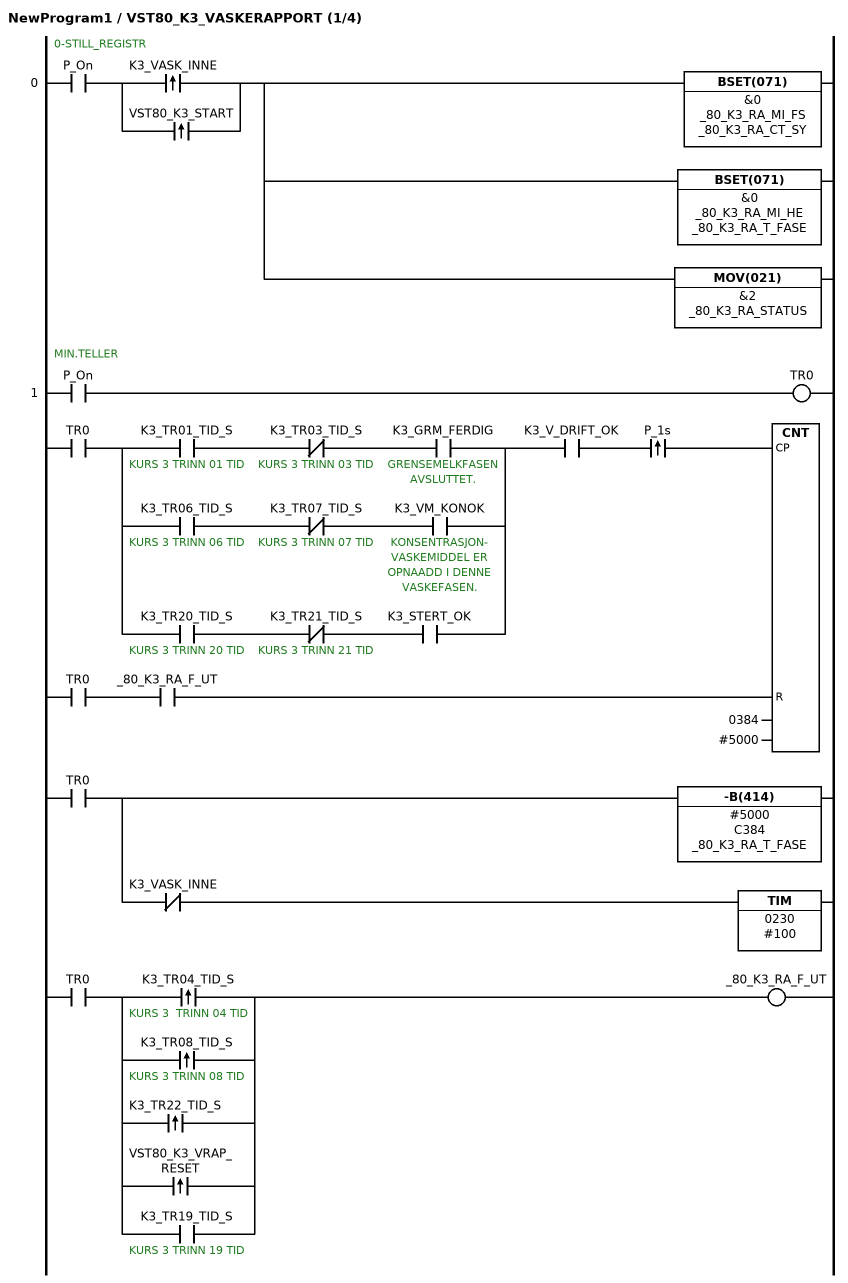
; [picture p384: NewProgram1 / VST80_K3_VASKERAPPORT, rungs 0-1]
; rung 0: 0-STILL_REGISTR
LD P_On
@LD K3_VASK_INNE
@OR VST80_K3_START
ANDLD
BSET(071) &0 _80_K3_RA_MI_FS _80_K3_RA_CT_SY
BSET(071) &0 _80_K3_RA_MI_HE _80_K3_RA_T_FASE
MOV(021) &2 _80_K3_RA_STATUS
; rung 1: MIN.TELLER
LD P_On
OUT TR0
LD K3_TR01_TID_S  ; KURS 3 TRINN 01 TID
ANDNOT K3_TR03_TID_S  ; KURS 3 TRINN 03 TID
AND K3_GRM_FERDIG  ; GRENSEMELKFASEN AVSLUTTET.
LD K3_TR06_TID_S  ; KURS 3 TRINN 06 TID
ANDNOT K3_TR07_TID_S  ; KURS 3 TRINN 07 TID
AND K3_VM_KONOK  ; KONSENTRASJON-VASKEMIDDEL ER OPNAADD I DENNE VASKEFASEN.
ORLD
LD K3_TR20_TID_S  ; KURS 3 TRINN 20 TID
ANDNOT K3_TR21_TID_S  ; KURS 3 TRINN 21 TID
AND K3_STERT_OK
ORLD
ANDLD
AND K3_V_DRIFT_OK
@AND P_1s
LD TR0
AND _80_K3_RA_F_UT
CNT 0384 #5000
LD TR0
-B(414) #5000 C384 _80_K3_RA_T_FASE
ANDNOT K3_VASK_INNE
TIM 0230 #100
LD TR0
@LD K3_TR04_TID_S  ; KURS 3  TRINN 04 TID
@OR K3_TR08_TID_S  ; KURS 3 TRINN 08 TID
@OR K3_TR22_TID_S
@OR VST80_K3_VRAP_RESET
OR K3_TR19_TID_S  ; KURS 3 TRINN 19 TID
ANDLD
OUT _80_K3_RA_F_UT

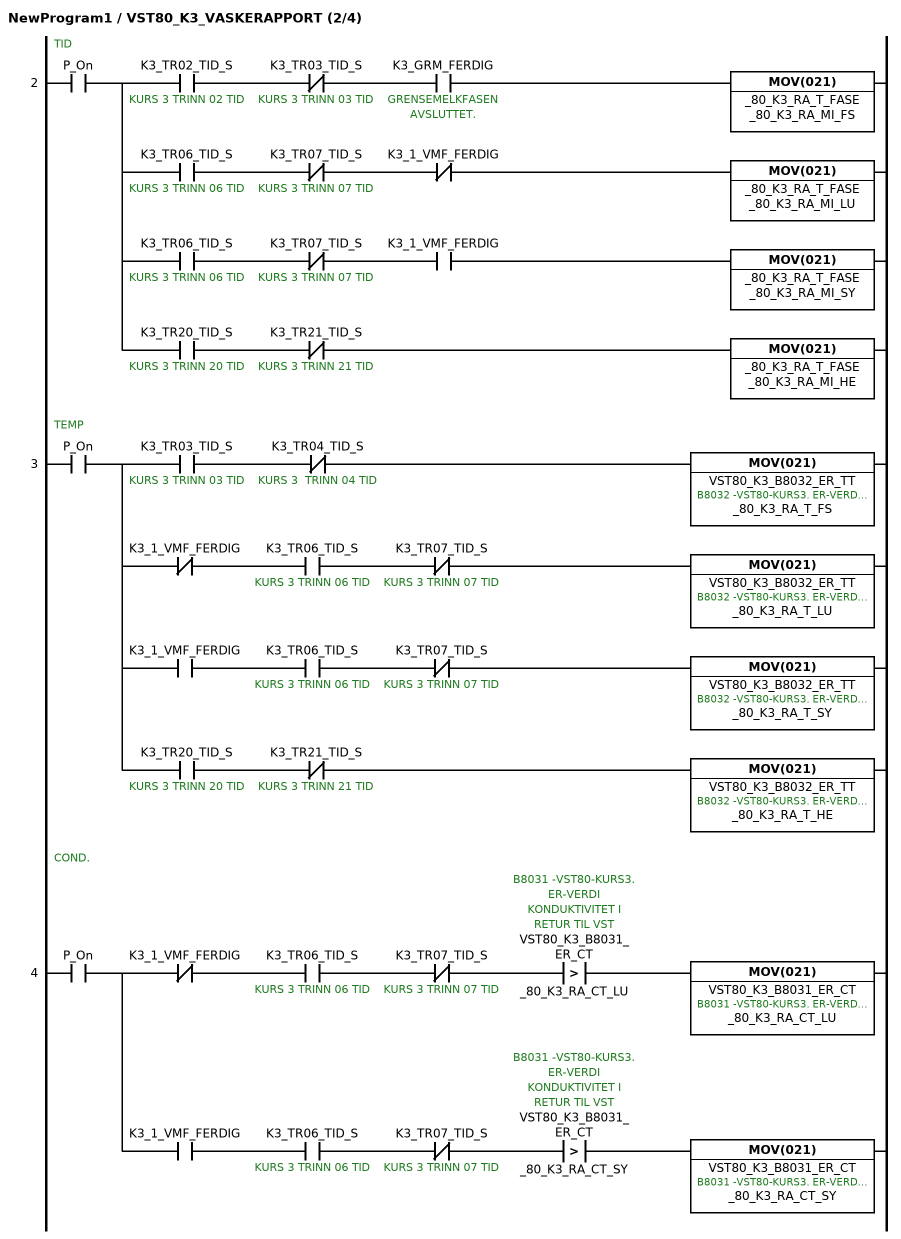
; rung 2: TID
LD P_On
OUT TR0
AND K3_TR02_TID_S  ; KURS 3 TRINN 02 TID
ANDNOT K3_TR03_TID_S  ; KURS 3 TRINN 03 TID
AND K3_GRM_FERDIG  ; GRENSEMELKFASEN AVSLUTTET.
MOV(021) _80_K3_RA_T_FASE _80_K3_RA_MI_FS
LD TR0
AND K3_TR06_TID_S  ; KURS 3 TRINN 06 TID
ANDNOT K3_TR07_TID_S  ; KURS 3 TRINN 07 TID
ANDNOT K3_1_VMF_FERDIG
MOV(021) _80_K3_RA_T_FASE _80_K3_RA_MI_LU
LD TR0
AND K3_TR06_TID_S  ; KURS 3 TRINN 06 TID
ANDNOT K3_TR07_TID_S  ; KURS 3 TRINN 07 TID
AND K3_1_VMF_FERDIG
MOV(021) _80_K3_RA_T_FASE _80_K3_RA_MI_SY
LD TR0
AND K3_TR20_TID_S  ; KURS 3 TRINN 20 TID
ANDNOT K3_TR21_TID_S  ; KURS 3 TRINN 21 TID
MOV(021) _80_K3_RA_T_FASE _80_K3_RA_MI_HE
; rung 3: TEMP
LD P_On
OUT TR0
AND K3_TR03_TID_S  ; KURS 3 TRINN 03 TID
ANDNOT K3_TR04_TID_S  ; KURS 3  TRINN 04 TID
MOV(021) VST80_K3_B8032_ER_TT _80_K3_RA_T_FS  ; B8032 -VST80-KURS3. ER-VERDI TEMPERATUR I RETUR TIL VST
LD TR0
ANDNOT K3_1_VMF_FERDIG
AND K3_TR06_TID_S  ; KURS 3 TRINN 06 TID
ANDNOT K3_TR07_TID_S  ; KURS 3 TRINN 07 TID
MOV(021) VST80_K3_B8032_ER_TT _80_K3_RA_T_LU  ; B8032 -VST80-KURS3. ER-VERDI TEMPERATUR I RETUR TIL VST
LD TR0
AND K3_1_VMF_FERDIG
AND K3_TR06_TID_S  ; KURS 3 TRINN 06 TID
ANDNOT K3_TR07_TID_S  ; KURS 3 TRINN 07 TID
MOV(021) VST80_K3_B8032_ER_TT _80_K3_RA_T_SY  ; B8032 -VST80-KURS3. ER-VERDI TEMPERATUR I RETUR TIL VST
LD TR0
AND K3_TR20_TID_S  ; KURS 3 TRINN 20 TID
ANDNOT K3_TR21_TID_S  ; KURS 3 TRINN 21 TID
MOV(021) VST80_K3_B8032_ER_TT _80_K3_RA_T_HE  ; B8032 -VST80-KURS3. ER-VERDI TEMPERATUR I RETUR TIL VST
; rung 4: COND.
LD P_On
OUT TR0
ANDNOT K3_1_VMF_FERDIG
AND K3_TR06_TID_S  ; KURS 3 TRINN 06 TID
ANDNOT K3_TR07_TID_S  ; KURS 3 TRINN 07 TID
AND>(320) VST80_K3_B8031_ER_CT _80_K3_RA_CT_LU  ; B8031 -VST80-KURS3. ER-VERDI KONDUKTIVITET I RETUR TIL VST
MOV(021) VST80_K3_B8031_ER_CT _80_K3_RA_CT_LU  ; B8031 -VST80-KURS3. ER-VERDI KONDUKTIVITET I RETUR TIL VST
LD TR0
AND K3_1_VMF_FERDIG
AND K3_TR06_TID_S  ; KURS 3 TRINN 06 TID
ANDNOT K3_TR07_TID_S  ; KURS 3 TRINN 07 TID
AND>(320) VST80_K3_B8031_ER_CT _80_K3_RA_CT_SY  ; B8031 -VST80-KURS3. ER-VERDI KONDUKTIVITET I RETUR TIL VST
MOV(021) VST80_K3_B8031_ER_CT _80_K3_RA_CT_SY  ; B8031 -VST80-KURS3. ER-VERDI KONDUKTIVITET I RETUR TIL VST

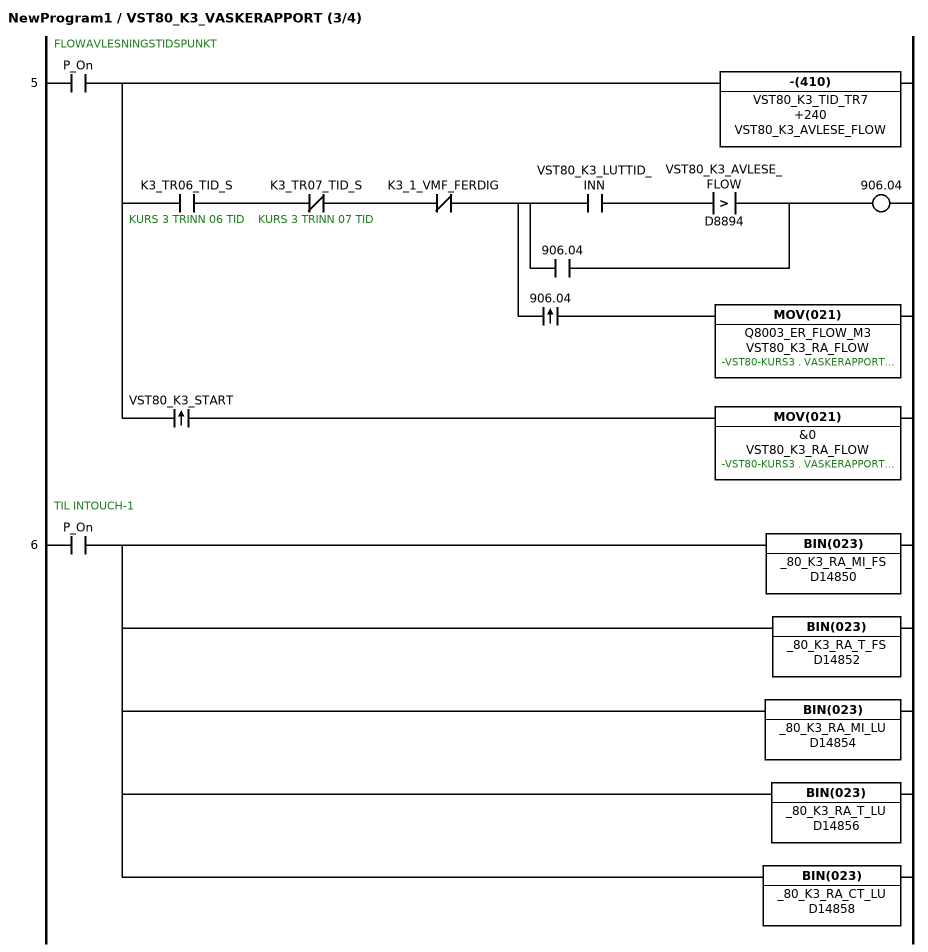
; rung 5: FLOWAVLESNINGSTIDSPUNKT
LD P_On
OUT TR0
-(410) VST80_K3_TID_TR7 +240 VST80_K3_AVLESE_FLOW
AND K3_TR06_TID_S  ; KURS 3 TRINN 06 TID
ANDNOT K3_TR07_TID_S  ; KURS 3 TRINN 07 TID
ANDNOT K3_1_VMF_FERDIG
OUT TR1
LD VST80_K3_LUTTID_INN
AND>(320) VST80_K3_AVLESE_FLOW D8894
OR 906.04
ANDLD
OUT 906.04
LD TR1
@AND 906.04
MOV(021) Q8003_ER_FLOW_M3 VST80_K3_RA_FLOW  ; -VST80-KURS3 . VASKERAPPORT.  FLOW
LD TR0
@AND VST80_K3_START
MOV(021) &0 VST80_K3_RA_FLOW  ; -VST80-KURS3 . VASKERAPPORT.  FLOW
; rung 6: TIL INTOUCH-1
LD P_On
BIN(023) _80_K3_RA_MI_FS D14850
BIN(023) _80_K3_RA_T_FS D14852
BIN(023) _80_K3_RA_MI_LU D14854
BIN(023) _80_K3_RA_T_LU D14856
BIN(023) _80_K3_RA_CT_LU D14858

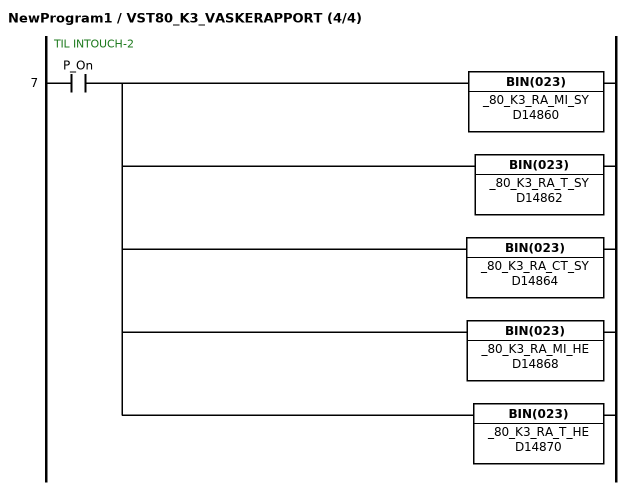
; rung 7: TIL INTOUCH-2
LD P_On
BIN(023) _80_K3_RA_MI_SY D14860
BIN(023) _80_K3_RA_T_SY D14862
BIN(023) _80_K3_RA_CT_SY D14864
BIN(023) _80_K3_RA_MI_HE D14868
BIN(023) _80_K3_RA_T_HE D14870
; rung 8: Ingen_kommentar_funnet

### Section VST80_K3_REGULATORER

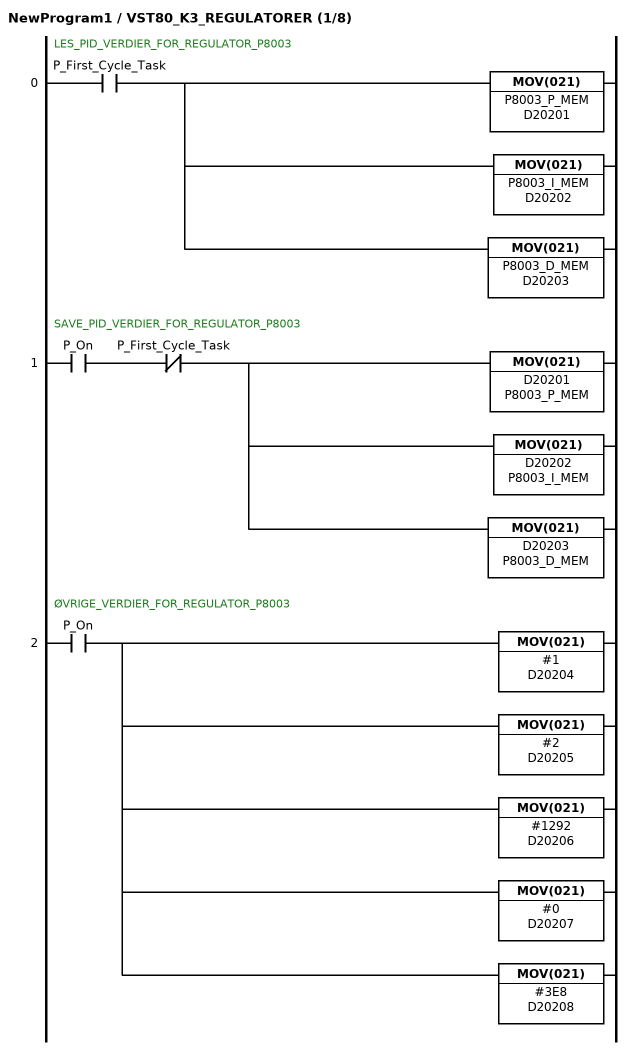
; rung 0: LES_PID_VERDIER_FOR_REGULATOR_P8003
LD P_First_Cycle_Task
MOV(021) P8003_P_MEM D20201
MOV(021) P8003_I_MEM D20202
MOV(021) P8003_D_MEM D20203
; rung 1: SAVE_PID_VERDIER_FOR_REGULATOR_P8003
LD P_On
ANDNOT P_First_Cycle_Task
MOV(021) D20201 P8003_P_MEM
MOV(021) D20202 P8003_I_MEM
MOV(021) D20203 P8003_D_MEM
; rung 2: ØVRIGE_VERDIER_FOR_REGULATOR_P8003
LD P_On
MOV(021) #1 D20204
MOV(021) #2 D20205
MOV(021) #1292 D20206
MOV(021) #0 D20207
MOV(021) #3E8 D20208

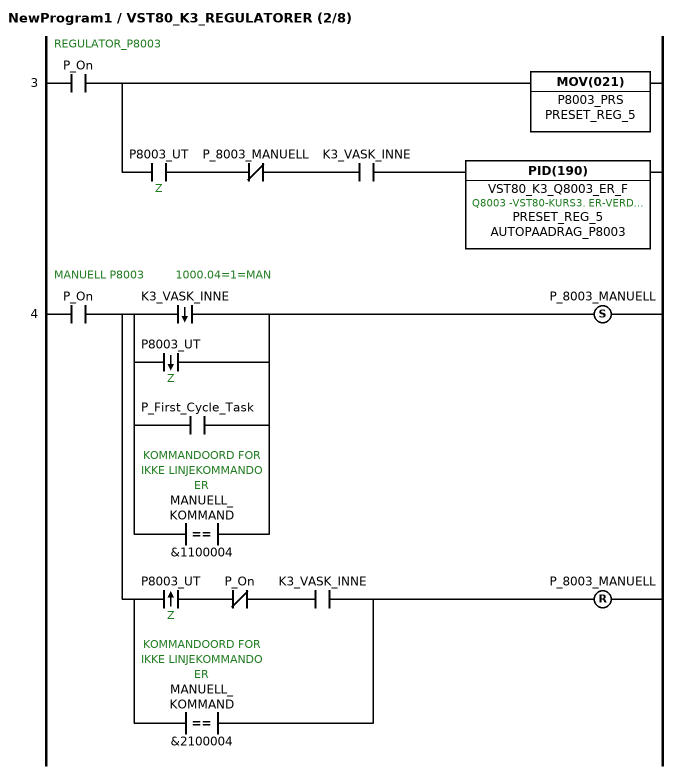
; rung 3: REGULATOR_P8003
LD P_On
MOV(021) P8003_PRS PRESET_REG_5
AND P8003_UT  ; Z
ANDNOT P_8003_MANUELL
AND K3_VASK_INNE
PID(190) VST80_K3_Q8003_ER_F PRESET_REG_5 AUTOPAADRAG_P8003  ; Q8003 -VST80-KURS3. ER-VERDI FLOW I TUR
; rung 4: MANUELL P8003         1000.04=1=MAN
LD P_On
OUT TR0
%LD K3_VASK_INNE
%OR P8003_UT  ; Z
OR P_First_Cycle_Task
OR=L(301) MANUELL_KOMMAND &1100004  ; KOMMANDOORD FOR IKKE LINJEKOMMANDOER
ANDLD
SET P_8003_MANUELL
LD TR0
@LD P8003_UT  ; Z
ANDNOT P_On
AND K3_VASK_INNE
OR=L(301) MANUELL_KOMMAND &2100004  ; KOMMANDOORD FOR IKKE LINJEKOMMANDOER
ANDLD
RSET P_8003_MANUELL

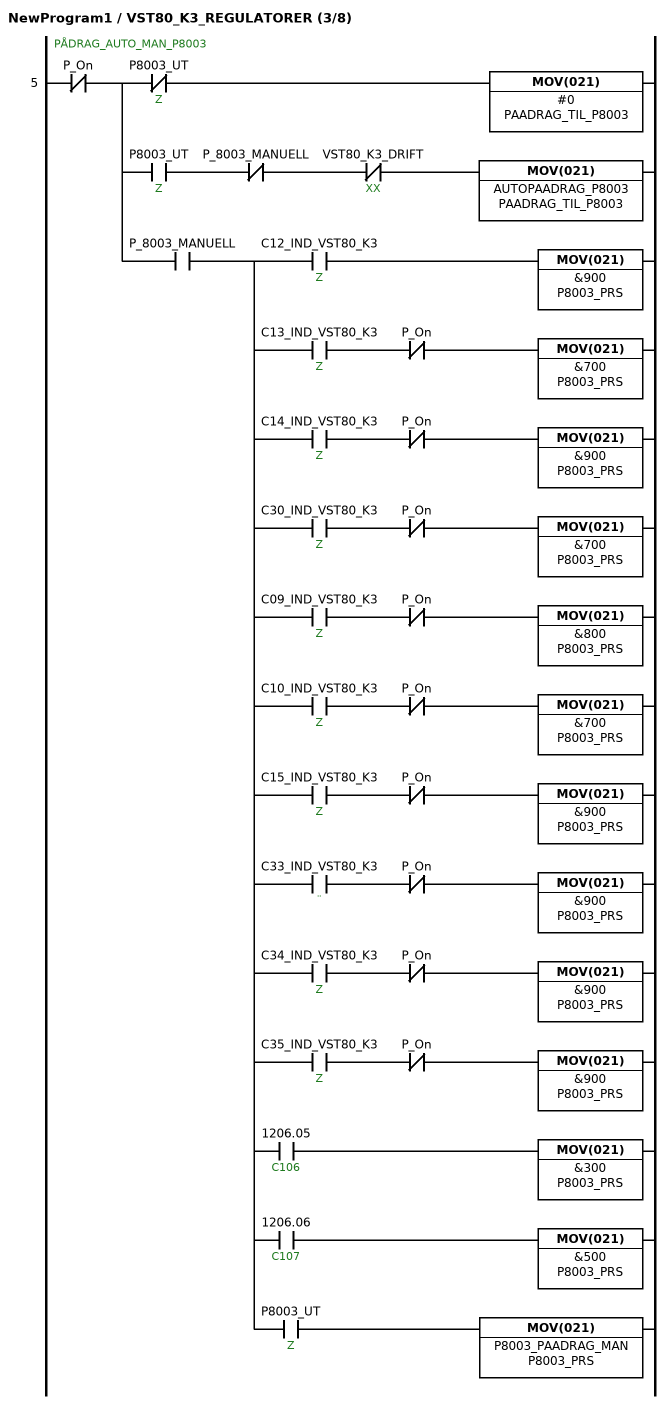
; rung 5: PÅDRAG_AUTO_MAN_P8003
LDNOT P_On
OUT TR0
ANDNOT P8003_UT  ; Z
MOV(021) #0 PAADRAG_TIL_P8003
LD TR0
AND P8003_UT  ; Z
ANDNOT P_8003_MANUELL
ANDNOT VST80_K3_DRIFT  ; XX
MOV(021) AUTOPAADRAG_P8003 PAADRAG_TIL_P8003
LD TR0
AND P_8003_MANUELL
OUT TR0
AND C12_IND_VST80_K3  ; Z
MOV(021) &900 P8003_PRS
LD TR0
AND C13_IND_VST80_K3  ; Z
ANDNOT P_On
MOV(021) &700 P8003_PRS
LD TR0
AND C14_IND_VST80_K3  ; Z
ANDNOT P_On
MOV(021) &900 P8003_PRS
LD TR0
AND C30_IND_VST80_K3  ; Z
ANDNOT P_On
MOV(021) &700 P8003_PRS
LD TR0
AND C09_IND_VST80_K3  ; Z
ANDNOT P_On
MOV(021) &800 P8003_PRS
LD TR0
AND C10_IND_VST80_K3  ; Z
ANDNOT P_On
MOV(021) &700 P8003_PRS
LD TR0
AND C15_IND_VST80_K3  ; Z
ANDNOT P_On
MOV(021) &900 P8003_PRS
LD TR0
AND C33_IND_VST80_K3  ; ¨
ANDNOT P_On
MOV(021) &900 P8003_PRS
LD TR0
AND C34_IND_VST80_K3  ; Z
ANDNOT P_On
MOV(021) &900 P8003_PRS
LD TR0
AND C35_IND_VST80_K3  ; Z
ANDNOT P_On
MOV(021) &900 P8003_PRS
LD TR0
AND 1206.05  ; C106
MOV(021) &300 P8003_PRS
LD TR0
AND 1206.06  ; C107
MOV(021) &500 P8003_PRS
LD TR0
AND P8003_UT  ; Z
MOV(021) P8003_PAADRAG_MAN P8003_PRS

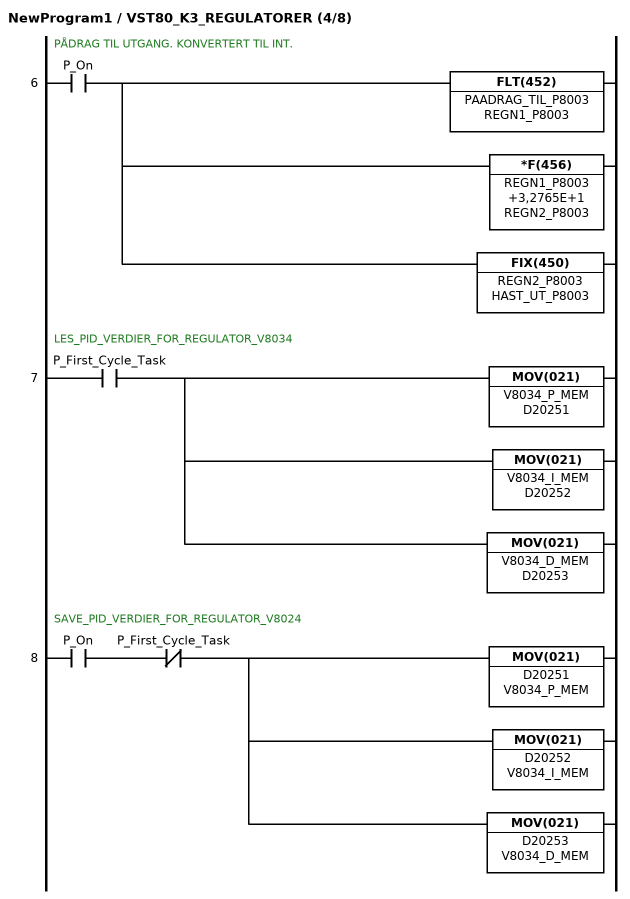
; rung 6: PÅDRAG TIL UTGANG. KONVERTERT TIL INT.
LD P_On
FLT(452) PAADRAG_TIL_P8003 REGN1_P8003
*F(456) REGN1_P8003 +3,2765E+1 REGN2_P8003
FIX(450) REGN2_P8003 HAST_UT_P8003
; rung 7: LES_PID_VERDIER_FOR_REGULATOR_V8034
LD P_First_Cycle_Task
MOV(021) V8034_P_MEM D20251
MOV(021) V8034_I_MEM D20252
MOV(021) V8034_D_MEM D20253
; rung 8: SAVE_PID_VERDIER_FOR_REGULATOR_V8024
LD P_On
ANDNOT P_First_Cycle_Task
MOV(021) D20251 V8034_P_MEM
MOV(021) D20252 V8034_I_MEM
MOV(021) D20253 V8034_D_MEM

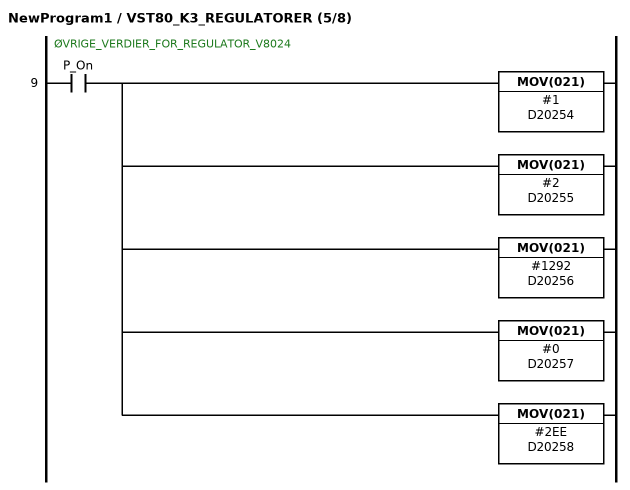
; rung 9: ØVRIGE_VERDIER_FOR_REGULATOR_V8024
LD P_On
MOV(021) #1 D20254
MOV(021) #2 D20255
MOV(021) #1292 D20256
MOV(021) #0 D20257
MOV(021) #2EE D20258

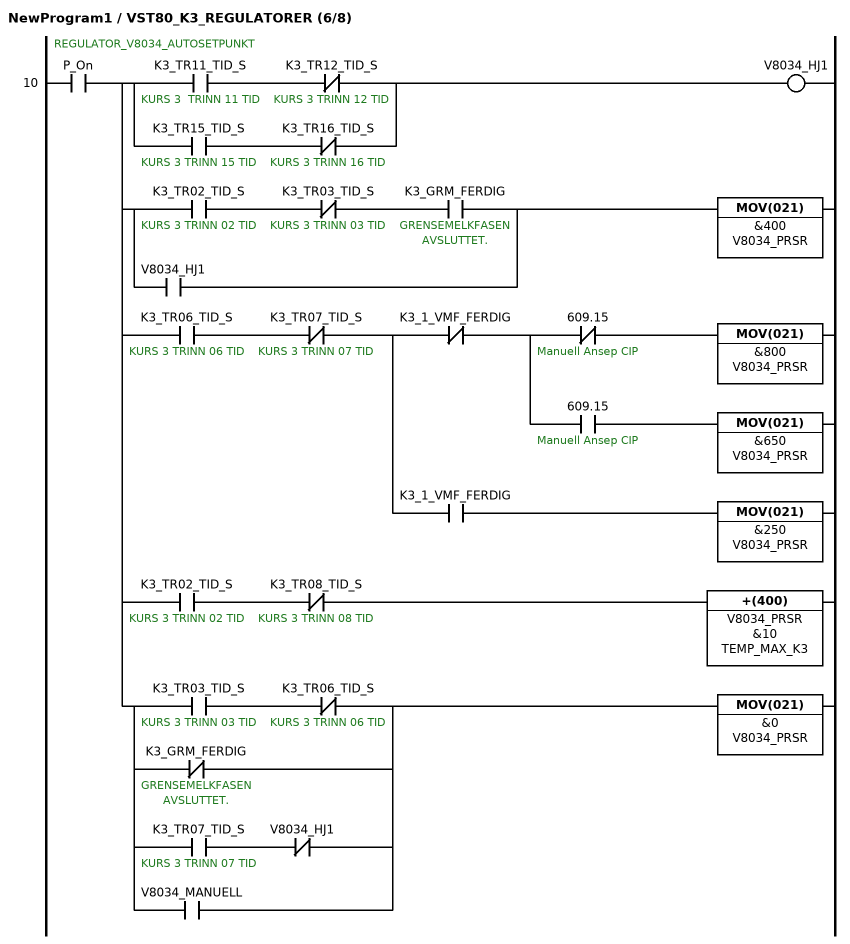
; rung 10: REGULATOR_V8034_AUTOSETPUNKT
LD P_On
OUT TR0
LD K3_TR11_TID_S  ; KURS 3  TRINN 11 TID
ANDNOT K3_TR12_TID_S  ; KURS 3 TRINN 12 TID
LD K3_TR15_TID_S  ; KURS 3 TRINN 15 TID
ANDNOT K3_TR16_TID_S  ; KURS 3 TRINN 16 TID
ORLD
ANDLD
OUT V8034_HJ1
LD TR0
LD K3_TR02_TID_S  ; KURS 3 TRINN 02 TID
ANDNOT K3_TR03_TID_S  ; KURS 3 TRINN 03 TID
AND K3_GRM_FERDIG  ; GRENSEMELKFASEN AVSLUTTET.
OR V8034_HJ1
ANDLD
MOV(021) &400 V8034_PRSR
LD TR0
AND K3_TR06_TID_S  ; KURS 3 TRINN 06 TID
ANDNOT K3_TR07_TID_S  ; KURS 3 TRINN 07 TID
OUT TR1
ANDNOT K3_1_VMF_FERDIG
OUT TR2
ANDNOT 609.15  ; Manuell Ansep CIP
MOV(021) &800 V8034_PRSR
LD TR2
AND 609.15  ; Manuell Ansep CIP
MOV(021) &650 V8034_PRSR
LD TR1
AND K3_1_VMF_FERDIG
MOV(021) &250 V8034_PRSR
LD TR0
AND K3_TR02_TID_S  ; KURS 3 TRINN 02 TID
ANDNOT K3_TR08_TID_S  ; KURS 3 TRINN 08 TID
+(400) V8034_PRSR &10 TEMP_MAX_K3
LD TR0
LD K3_TR03_TID_S  ; KURS 3 TRINN 03 TID
ANDNOT K3_TR06_TID_S  ; KURS 3 TRINN 06 TID
ORNOT K3_GRM_FERDIG  ; GRENSEMELKFASEN AVSLUTTET.
LD K3_TR07_TID_S  ; KURS 3 TRINN 07 TID
ANDNOT V8034_HJ1
ORLD
OR V8034_MANUELL
ANDLD
MOV(021) &0 V8034_PRSR

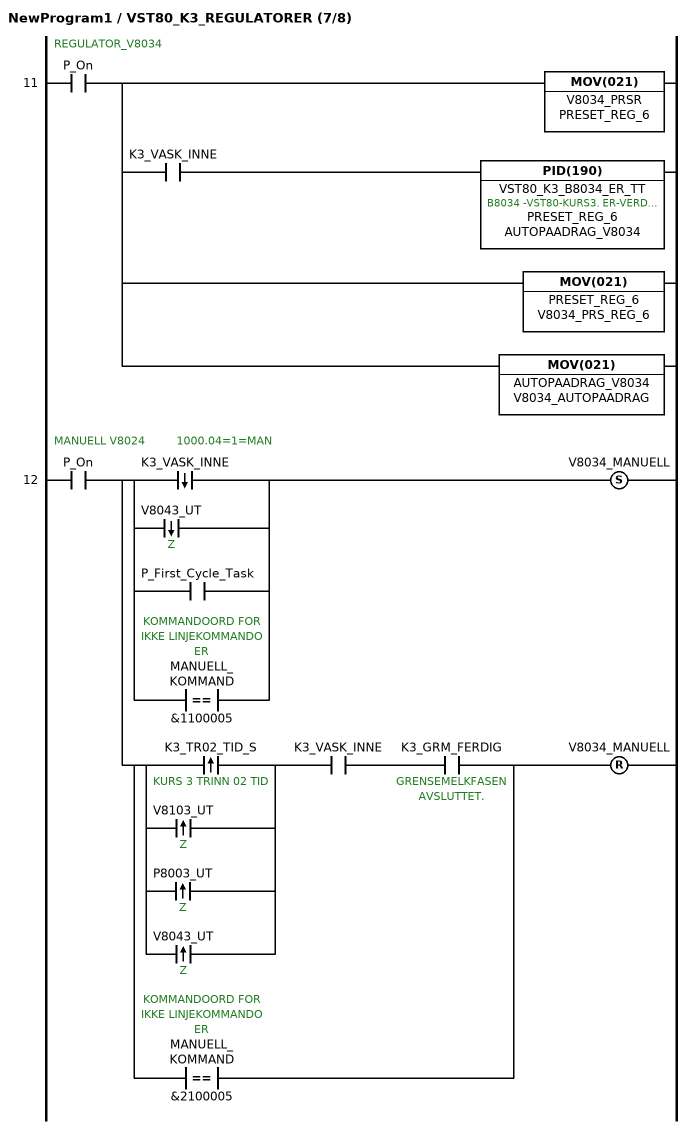
; rung 11: REGULATOR_V8034
LD P_On
OUT TR0
MOV(021) V8034_PRSR PRESET_REG_6
AND K3_VASK_INNE
PID(190) VST80_K3_B8034_ER_TT PRESET_REG_6 AUTOPAADRAG_V8034  ; B8034 -VST80-KURS3. ER-VERDI TEMPERATUR I TUR TIL VST
LD TR0
MOV(021) PRESET_REG_6 V8034_PRS_REG_6
MOV(021) AUTOPAADRAG_V8034 V8034_AUTOPAADRAG
; rung 12: MANUELL V8024         1000.04=1=MAN
LD P_On
OUT TR0
%LD K3_VASK_INNE
%OR V8043_UT  ; Z
OR P_First_Cycle_Task
OR=L(301) MANUELL_KOMMAND &1100005  ; KOMMANDOORD FOR IKKE LINJEKOMMANDOER
ANDLD
SET V8034_MANUELL
LD TR0
@LD K3_TR02_TID_S  ; KURS 3 TRINN 02 TID
@OR V8103_UT  ; Z
@OR P8003_UT  ; Z
@OR V8043_UT  ; Z
AND K3_VASK_INNE
AND K3_GRM_FERDIG  ; GRENSEMELKFASEN AVSLUTTET.
OR=L(301) MANUELL_KOMMAND &2100005  ; KOMMANDOORD FOR IKKE LINJEKOMMANDOER
ANDLD
RSET V8034_MANUELL

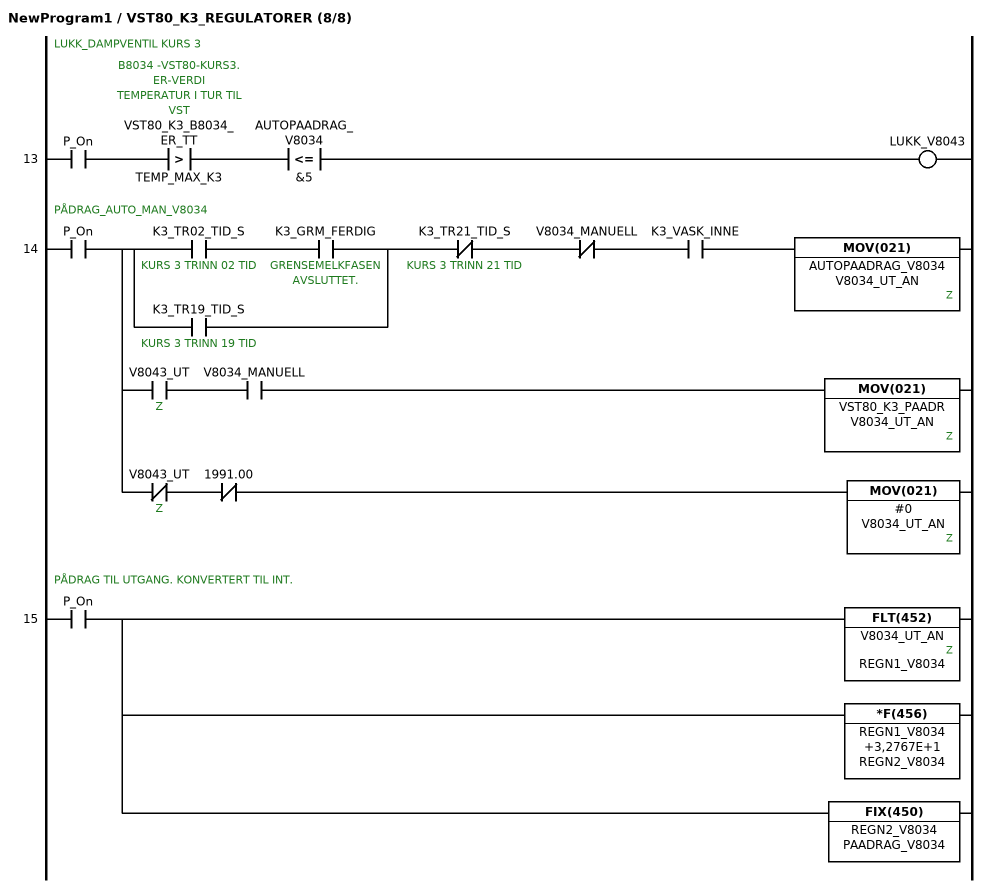
; rung 13: LUKK_DAMPVENTIL KURS 3
LD P_On
AND>(320) VST80_K3_B8034_ER_TT TEMP_MAX_K3  ; B8034 -VST80-KURS3. ER-VERDI TEMPERATUR I TUR TIL VST
AND<=(315) AUTOPAADRAG_V8034 &5
OUT LUKK_V8043
; rung 14: PÅDRAG_AUTO_MAN_V8034
LD P_On
OUT TR0
LD K3_TR02_TID_S  ; KURS 3 TRINN 02 TID
AND K3_GRM_FERDIG  ; GRENSEMELKFASEN AVSLUTTET.
OR K3_TR19_TID_S  ; KURS 3 TRINN 19 TID
ANDLD
ANDNOT K3_TR21_TID_S  ; KURS 3 TRINN 21 TID
ANDNOT V8034_MANUELL
AND K3_VASK_INNE
MOV(021) AUTOPAADRAG_V8034 V8034_UT_AN  ; Z
LD TR0
AND V8043_UT  ; Z
AND V8034_MANUELL
MOV(021) VST80_K3_PAADR V8034_UT_AN  ; Z
LD TR0
ANDNOT V8043_UT  ; Z
ANDNOT 1991.00
MOV(021) #0 V8034_UT_AN  ; Z
; rung 15: PÅDRAG TIL UTGANG. KONVERTERT TIL INT.
LD P_On
FLT(452) V8034_UT_AN REGN1_V8034  ; Z
*F(456) REGN1_V8034 +3,2767E+1 REGN2_V8034
FIX(450) REGN2_V8034 PAADRAG_V8034
; rung 16: Ingen_kommentar_funnet

### Section VST80_AUTOVASK_KURS_3

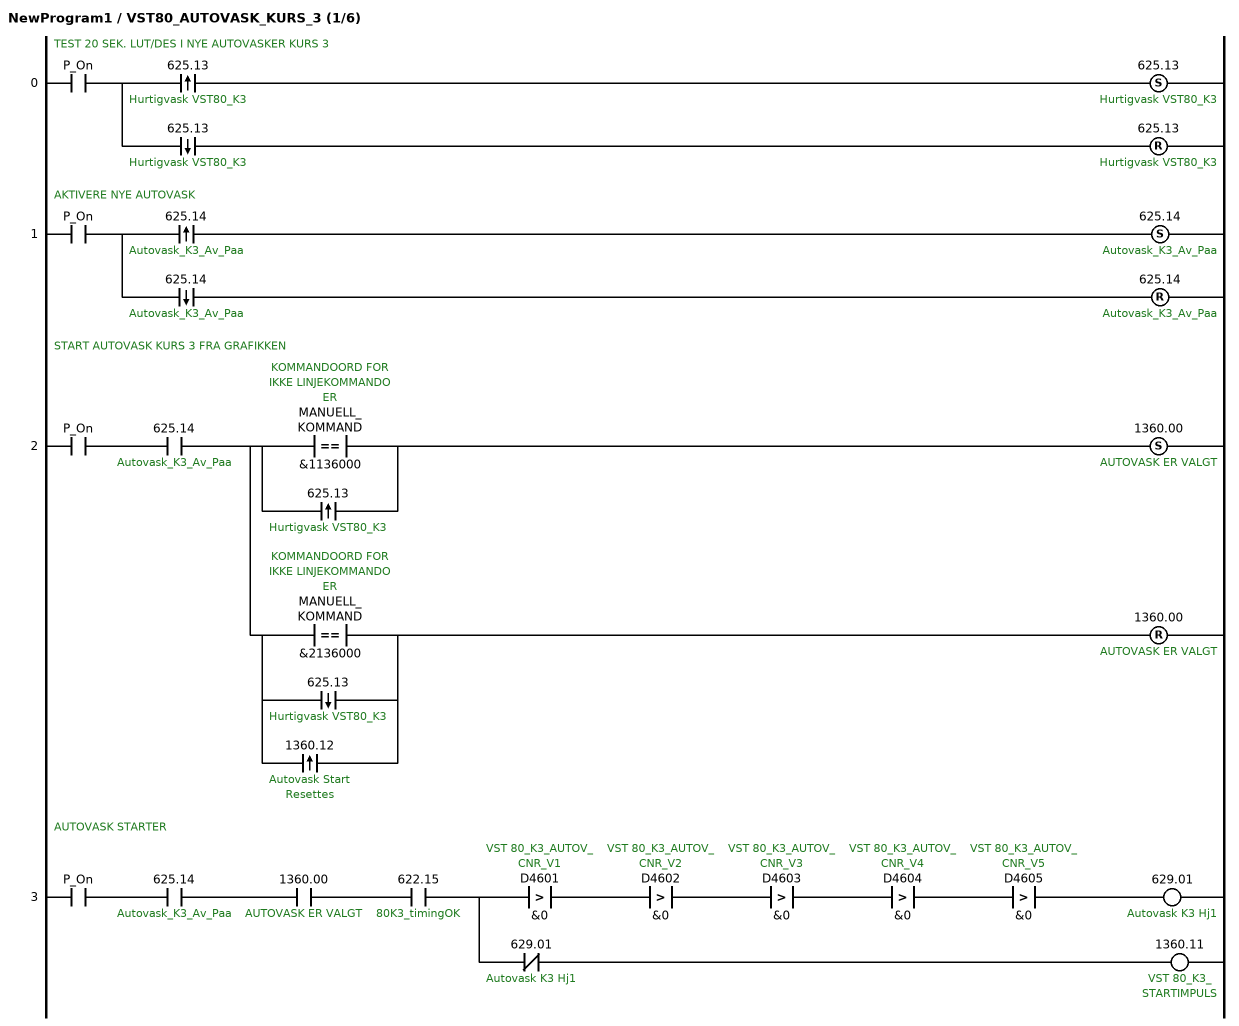
; rung 0: TEST 20 SEK. LUT/DES I NYE AUTOVASKER KURS 3
LD P_On
OUT TR0
@AND 625.13  ; Hurtigvask VST80_K3
SET 625.13  ; Hurtigvask VST80_K3
LD TR0
%AND 625.13  ; Hurtigvask VST80_K3
RSET 625.13  ; Hurtigvask VST80_K3
; rung 1: AKTIVERE NYE AUTOVASK
LD P_On
OUT TR0
@AND 625.14  ; Autovask_K3_Av_Paa
SET 625.14  ; Autovask_K3_Av_Paa
LD TR0
%AND 625.14  ; Autovask_K3_Av_Paa
RSET 625.14  ; Autovask_K3_Av_Paa
; rung 2: START AUTOVASK KURS 3 FRA GRAFIKKEN
LD P_On
AND 625.14  ; Autovask_K3_Av_Paa
OUT TR0
LD=L(301) MANUELL_KOMMAND &1136000  ; KOMMANDOORD FOR IKKE LINJEKOMMANDOER
@OR 625.13  ; Hurtigvask VST80_K3
ANDLD
SET 1360.00  ; AUTOVASK ER VALGT
LD TR0
LD=L(301) MANUELL_KOMMAND &2136000  ; KOMMANDOORD FOR IKKE LINJEKOMMANDOER
%OR 625.13  ; Hurtigvask VST80_K3
@OR 1360.12  ; Autovask Start Resettes
ANDLD
RSET 1360.00  ; AUTOVASK ER VALGT
; rung 3: AUTOVASK STARTER
LD P_On
AND 625.14  ; Autovask_K3_Av_Paa
AND 1360.00  ; AUTOVASK ER VALGT
AND 622.15  ; 80K3_timingOK
OUT TR0
AND>(320) D4601 &0  ; VST 80_K3_AUTOV_CNR_V1
AND>(320) D4602 &0  ; VST 80_K3_AUTOV_CNR_V2
AND>(320) D4603 &0  ; VST 80_K3_AUTOV_CNR_V3
AND>(320) D4604 &0  ; VST 80_K3_AUTOV_CNR_V4
AND>(320) D4605 &0  ; VST 80_K3_AUTOV_CNR_V5
OUT 629.01  ; Autovask K3 Hj1
LD TR0
ANDNOT 629.01  ; Autovask K3 Hj1
OUT 1360.11  ; VST 80_K3_STARTIMPULS

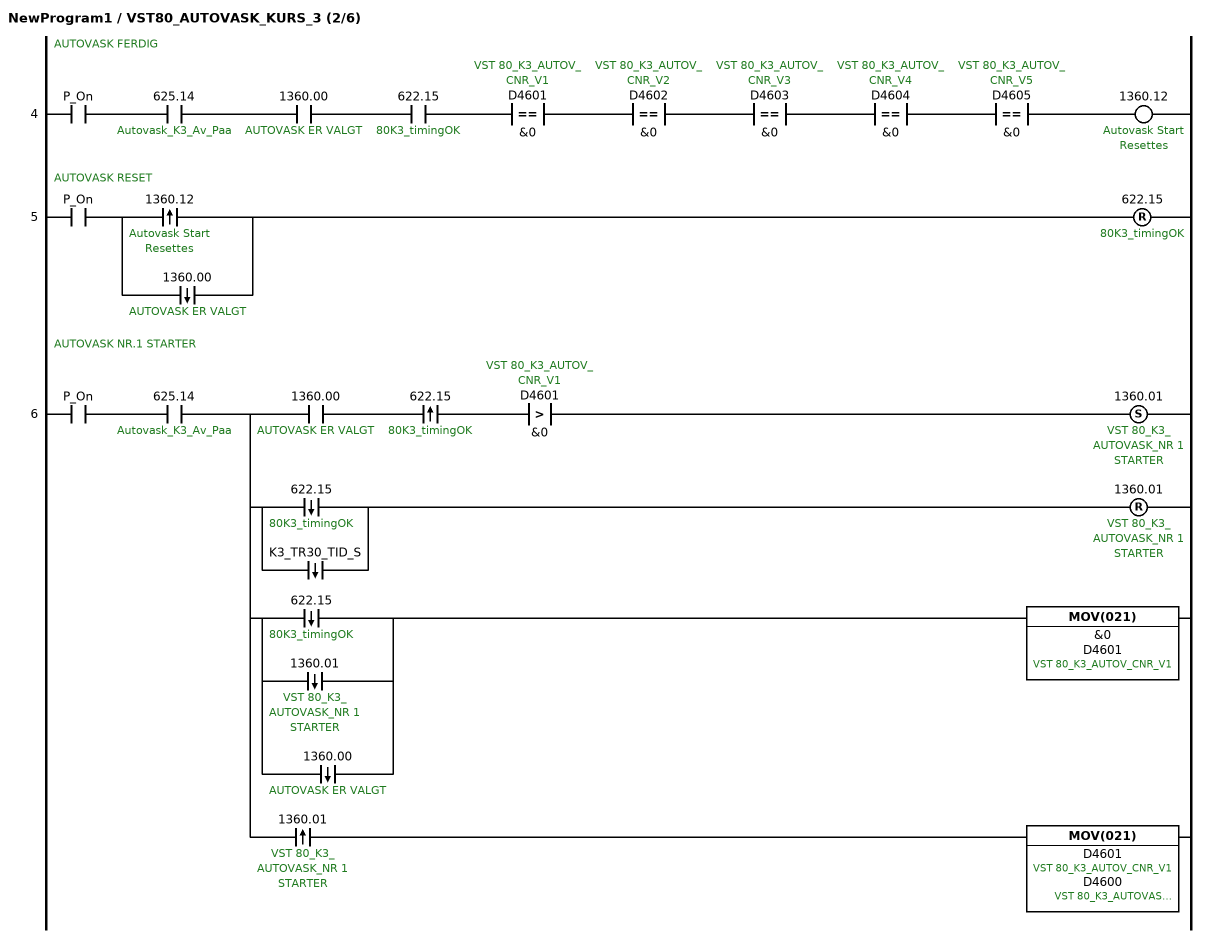
; rung 4: AUTOVASK FERDIG
LD P_On
AND 625.14  ; Autovask_K3_Av_Paa
AND 1360.00  ; AUTOVASK ER VALGT
AND 622.15  ; 80K3_timingOK
AND=(300) D4601 &0  ; VST 80_K3_AUTOV_CNR_V1
AND=(300) D4602 &0  ; VST 80_K3_AUTOV_CNR_V2
AND=(300) D4603 &0  ; VST 80_K3_AUTOV_CNR_V3
AND=(300) D4604 &0  ; VST 80_K3_AUTOV_CNR_V4
AND=(300) D4605 &0  ; VST 80_K3_AUTOV_CNR_V5
OUT 1360.12  ; Autovask Start Resettes
; rung 5: AUTOVASK RESET
LD P_On
@LD 1360.12  ; Autovask Start Resettes
%OR 1360.00  ; AUTOVASK ER VALGT
ANDLD
RSET 622.15  ; 80K3_timingOK
; rung 6: AUTOVASK NR.1 STARTER
LD P_On
AND 625.14  ; Autovask_K3_Av_Paa
OUT TR0
AND 1360.00  ; AUTOVASK ER VALGT
@AND 622.15  ; 80K3_timingOK
AND>(320) D4601 &0  ; VST 80_K3_AUTOV_CNR_V1
SET 1360.01  ; VST 80_K3_AUTOVASK_NR 1 STARTER
LD TR0
%LD 622.15  ; 80K3_timingOK
%OR K3_TR30_TID_S
ANDLD
RSET 1360.01  ; VST 80_K3_AUTOVASK_NR 1 STARTER
LD TR0
%LD 622.15  ; 80K3_timingOK
%OR 1360.01  ; VST 80_K3_AUTOVASK_NR 1 STARTER
%OR 1360.00  ; AUTOVASK ER VALGT
ANDLD
MOV(021) &0 D4601  ; VST 80_K3_AUTOV_CNR_V1
LD TR0
@AND 1360.01  ; VST 80_K3_AUTOVASK_NR 1 STARTER
MOV(021) D4601 D4600  ; VST 80_K3_AUTOV_CNR_V1, VST 80_K3_AUTOVASK FELLESREGISTER

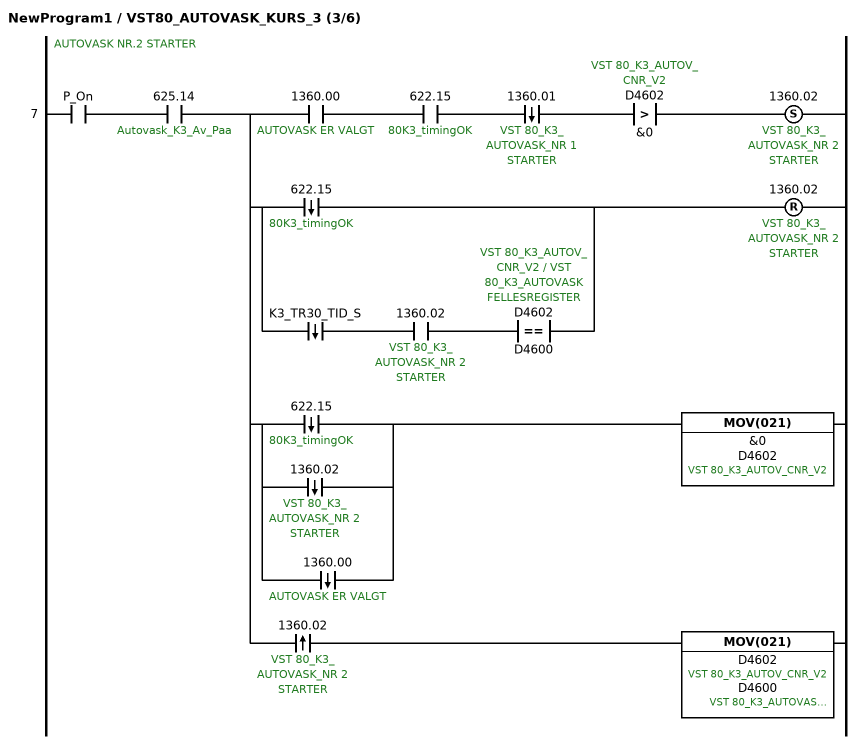
; rung 7: AUTOVASK NR.2 STARTER
LD P_On
AND 625.14  ; Autovask_K3_Av_Paa
OUT TR0
AND 1360.00  ; AUTOVASK ER VALGT
AND 622.15  ; 80K3_timingOK
%AND 1360.01  ; VST 80_K3_AUTOVASK_NR 1 STARTER
AND>(320) D4602 &0  ; VST 80_K3_AUTOV_CNR_V2
SET 1360.02  ; VST 80_K3_AUTOVASK_NR 2 STARTER
LD TR0
%LD 622.15  ; 80K3_timingOK
%LD K3_TR30_TID_S
AND 1360.02  ; VST 80_K3_AUTOVASK_NR 2 STARTER
AND=(300) D4602 D4600  ; VST 80_K3_AUTOV_CNR_V2, VST 80_K3_AUTOVASK FELLESREGISTER
ORLD
ANDLD
RSET 1360.02  ; VST 80_K3_AUTOVASK_NR 2 STARTER
LD TR0
%LD 622.15  ; 80K3_timingOK
%OR 1360.02  ; VST 80_K3_AUTOVASK_NR 2 STARTER
%OR 1360.00  ; AUTOVASK ER VALGT
ANDLD
MOV(021) &0 D4602  ; VST 80_K3_AUTOV_CNR_V2
LD TR0
@AND 1360.02  ; VST 80_K3_AUTOVASK_NR 2 STARTER
MOV(021) D4602 D4600  ; VST 80_K3_AUTOV_CNR_V2, VST 80_K3_AUTOVASK FELLESREGISTER

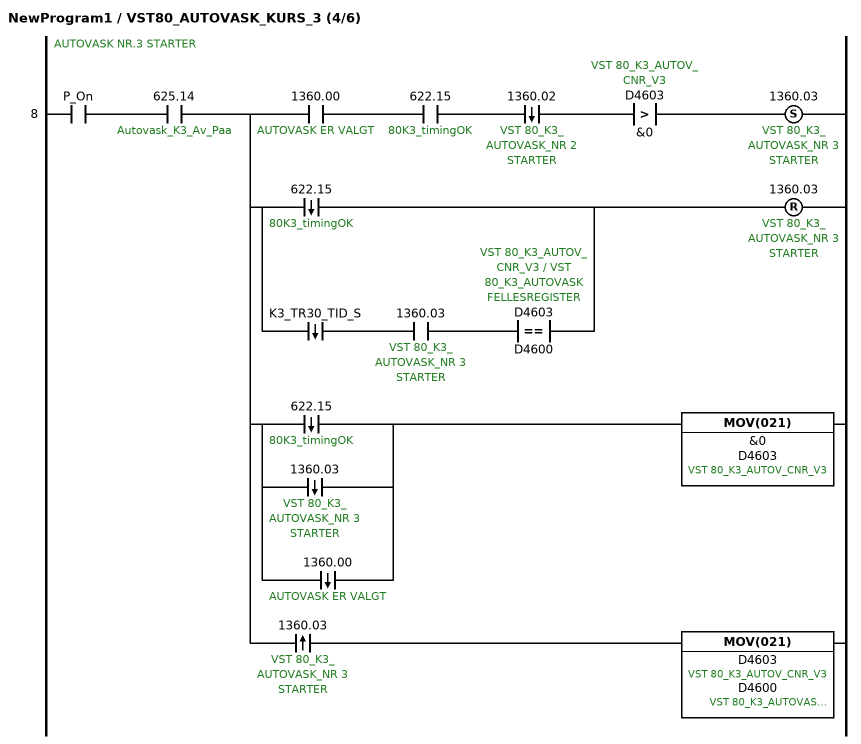
; rung 8: AUTOVASK NR.3 STARTER
LD P_On
AND 625.14  ; Autovask_K3_Av_Paa
OUT TR0
AND 1360.00  ; AUTOVASK ER VALGT
AND 622.15  ; 80K3_timingOK
%AND 1360.02  ; VST 80_K3_AUTOVASK_NR 2 STARTER
AND>(320) D4603 &0  ; VST 80_K3_AUTOV_CNR_V3
SET 1360.03  ; VST 80_K3_AUTOVASK_NR 3 STARTER
LD TR0
%LD 622.15  ; 80K3_timingOK
%LD K3_TR30_TID_S
AND 1360.03  ; VST 80_K3_AUTOVASK_NR 3 STARTER
AND=(300) D4603 D4600  ; VST 80_K3_AUTOV_CNR_V3, VST 80_K3_AUTOVASK FELLESREGISTER
ORLD
ANDLD
RSET 1360.03  ; VST 80_K3_AUTOVASK_NR 3 STARTER
LD TR0
%LD 622.15  ; 80K3_timingOK
%OR 1360.03  ; VST 80_K3_AUTOVASK_NR 3 STARTER
%OR 1360.00  ; AUTOVASK ER VALGT
ANDLD
MOV(021) &0 D4603  ; VST 80_K3_AUTOV_CNR_V3
LD TR0
@AND 1360.03  ; VST 80_K3_AUTOVASK_NR 3 STARTER
MOV(021) D4603 D4600  ; VST 80_K3_AUTOV_CNR_V3, VST 80_K3_AUTOVASK FELLESREGISTER

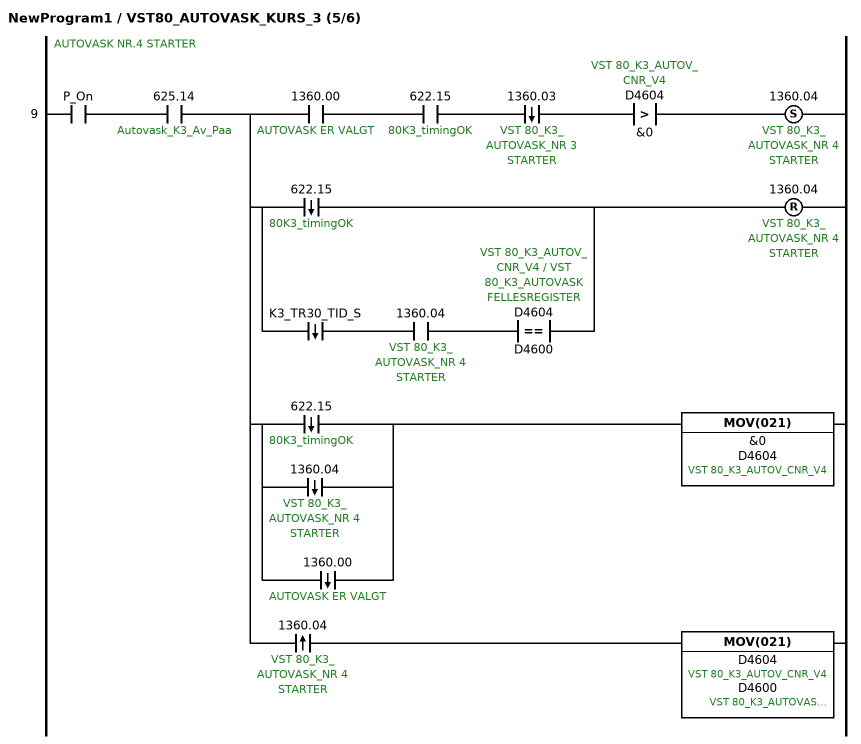
; rung 9: AUTOVASK NR.4 STARTER
LD P_On
AND 625.14  ; Autovask_K3_Av_Paa
OUT TR0
AND 1360.00  ; AUTOVASK ER VALGT
AND 622.15  ; 80K3_timingOK
%AND 1360.03  ; VST 80_K3_AUTOVASK_NR 3 STARTER
AND>(320) D4604 &0  ; VST 80_K3_AUTOV_CNR_V4
SET 1360.04  ; VST 80_K3_AUTOVASK_NR 4  STARTER
LD TR0
%LD 622.15  ; 80K3_timingOK
%LD K3_TR30_TID_S
AND 1360.04  ; VST 80_K3_AUTOVASK_NR 4  STARTER
AND=(300) D4604 D4600  ; VST 80_K3_AUTOV_CNR_V4, VST 80_K3_AUTOVASK FELLESREGISTER
ORLD
ANDLD
RSET 1360.04  ; VST 80_K3_AUTOVASK_NR 4  STARTER
LD TR0
%LD 622.15  ; 80K3_timingOK
%OR 1360.04  ; VST 80_K3_AUTOVASK_NR 4  STARTER
%OR 1360.00  ; AUTOVASK ER VALGT
ANDLD
MOV(021) &0 D4604  ; VST 80_K3_AUTOV_CNR_V4
LD TR0
@AND 1360.04  ; VST 80_K3_AUTOVASK_NR 4  STARTER
MOV(021) D4604 D4600  ; VST 80_K3_AUTOV_CNR_V4, VST 80_K3_AUTOVASK FELLESREGISTER

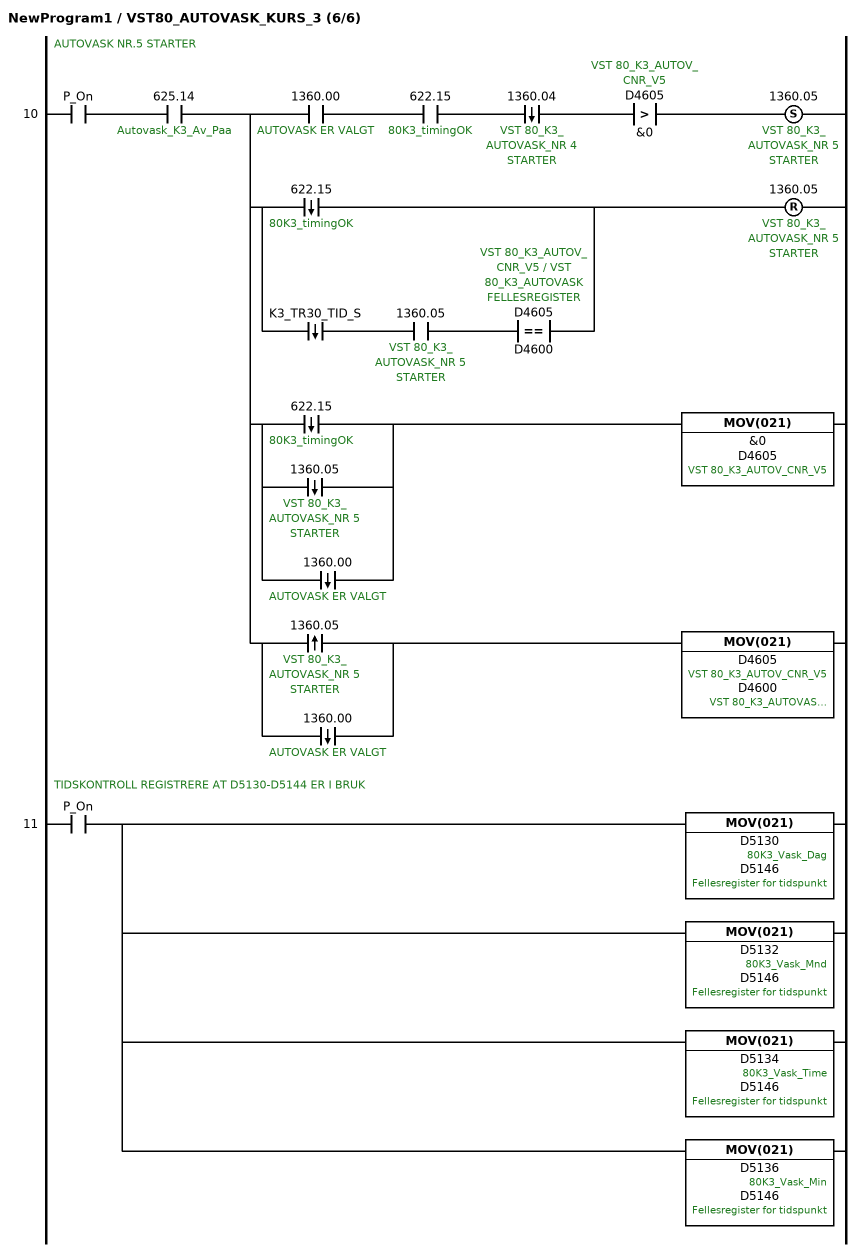
; rung 10: AUTOVASK NR.5 STARTER
LD P_On
AND 625.14  ; Autovask_K3_Av_Paa
OUT TR0
AND 1360.00  ; AUTOVASK ER VALGT
AND 622.15  ; 80K3_timingOK
%AND 1360.04  ; VST 80_K3_AUTOVASK_NR 4  STARTER
AND>(320) D4605 &0  ; VST 80_K3_AUTOV_CNR_V5
SET 1360.05  ; VST 80_K3_AUTOVASK_NR 5 STARTER
LD TR0
%LD 622.15  ; 80K3_timingOK
%LD K3_TR30_TID_S
AND 1360.05  ; VST 80_K3_AUTOVASK_NR 5 STARTER
AND=(300) D4605 D4600  ; VST 80_K3_AUTOV_CNR_V5, VST 80_K3_AUTOVASK FELLESREGISTER
ORLD
ANDLD
RSET 1360.05  ; VST 80_K3_AUTOVASK_NR 5 STARTER
LD TR0
%LD 622.15  ; 80K3_timingOK
%OR 1360.05  ; VST 80_K3_AUTOVASK_NR 5 STARTER
%OR 1360.00  ; AUTOVASK ER VALGT
ANDLD
MOV(021) &0 D4605  ; VST 80_K3_AUTOV_CNR_V5
LD TR0
@LD 1360.05  ; VST 80_K3_AUTOVASK_NR 5 STARTER
%OR 1360.00  ; AUTOVASK ER VALGT
ANDLD
MOV(021) D4605 D4600  ; VST 80_K3_AUTOV_CNR_V5, VST 80_K3_AUTOVASK FELLESREGISTER
; rung 11: TIDSKONTROLL REGISTRERE AT D5130-D5144 ER I BRUK
LD P_On
MOV(021) D5130 D5146  ; 80K3_Vask_Dag, Fellesregister for tidspunkt
MOV(021) D5132 D5146  ; 80K3_Vask_Mnd, Fellesregister for tidspunkt
MOV(021) D5134 D5146  ; 80K3_Vask_Time, Fellesregister for tidspunkt
MOV(021) D5136 D5146  ; 80K3_Vask_Min, Fellesregister for tidspunkt
; rung 12: Ingen_kommentar_funnet

### Section C23_FUNKSJONER

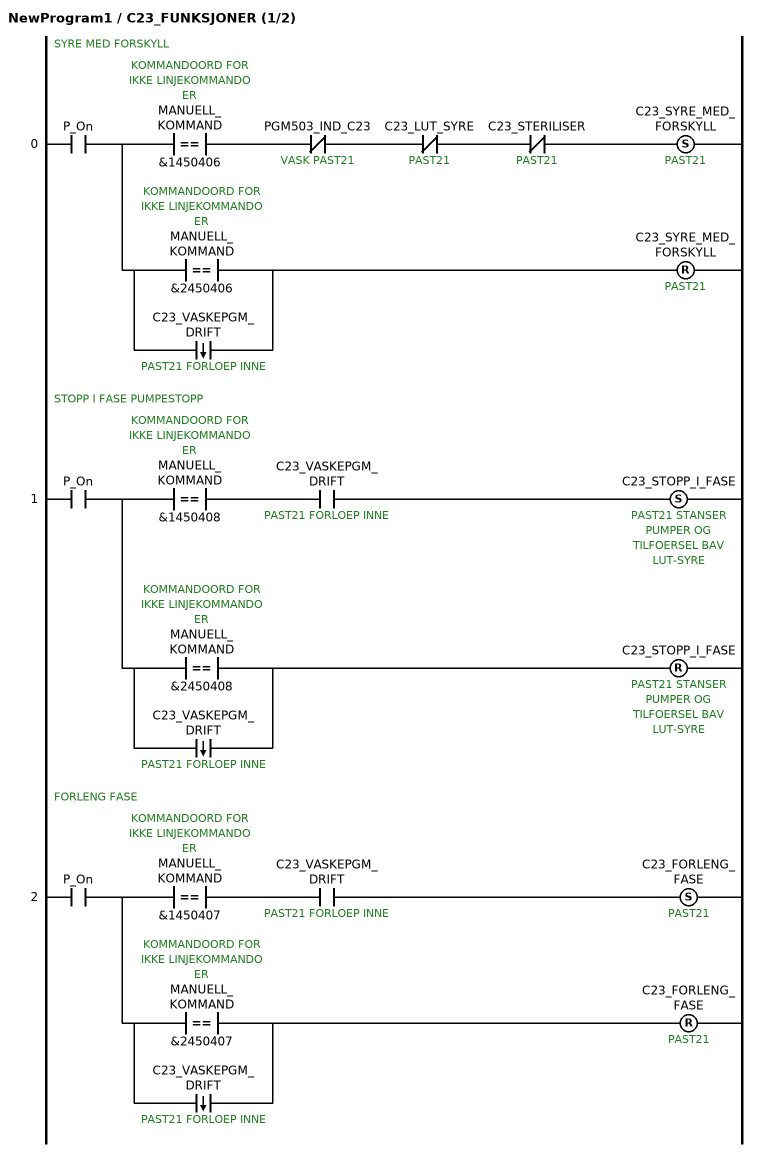
; rung 0: SYRE MED FORSKYLL
LD P_On
OUT TR0
AND=L(301) MANUELL_KOMMAND &1450406  ; KOMMANDOORD FOR IKKE LINJEKOMMANDOER
ANDNOT PGM503_IND_C23  ; VASK PAST21
ANDNOT C23_LUT_SYRE  ; PAST21
ANDNOT C23_STERILISER  ; PAST21
SET C23_SYRE_MED_FORSKYLL  ; PAST21
LD TR0
LD=L(301) MANUELL_KOMMAND &2450406  ; KOMMANDOORD FOR IKKE LINJEKOMMANDOER
%OR C23_VASKEPGM_DRIFT  ; PAST21 FORLOEP INNE
ANDLD
RSET C23_SYRE_MED_FORSKYLL  ; PAST21
; rung 1: STOPP I FASE PUMPESTOPP
LD P_On
OUT TR0
AND=L(301) MANUELL_KOMMAND &1450408  ; KOMMANDOORD FOR IKKE LINJEKOMMANDOER
AND C23_VASKEPGM_DRIFT  ; PAST21 FORLOEP INNE
SET C23_STOPP_I_FASE  ; PAST21 STANSER PUMPER OG TILFOERSEL BAV LUT-SYRE
LD TR0
LD=L(301) MANUELL_KOMMAND &2450408  ; KOMMANDOORD FOR IKKE LINJEKOMMANDOER
%OR C23_VASKEPGM_DRIFT  ; PAST21 FORLOEP INNE
ANDLD
RSET C23_STOPP_I_FASE  ; PAST21 STANSER PUMPER OG TILFOERSEL BAV LUT-SYRE
; rung 2: FORLENG FASE
LD P_On
OUT TR0
AND=L(301) MANUELL_KOMMAND &1450407  ; KOMMANDOORD FOR IKKE LINJEKOMMANDOER
AND C23_VASKEPGM_DRIFT  ; PAST21 FORLOEP INNE
SET C23_FORLENG_FASE  ; PAST21
LD TR0
LD=L(301) MANUELL_KOMMAND &2450407  ; KOMMANDOORD FOR IKKE LINJEKOMMANDOER
%OR C23_VASKEPGM_DRIFT  ; PAST21 FORLOEP INNE
ANDLD
RSET C23_FORLENG_FASE  ; PAST21

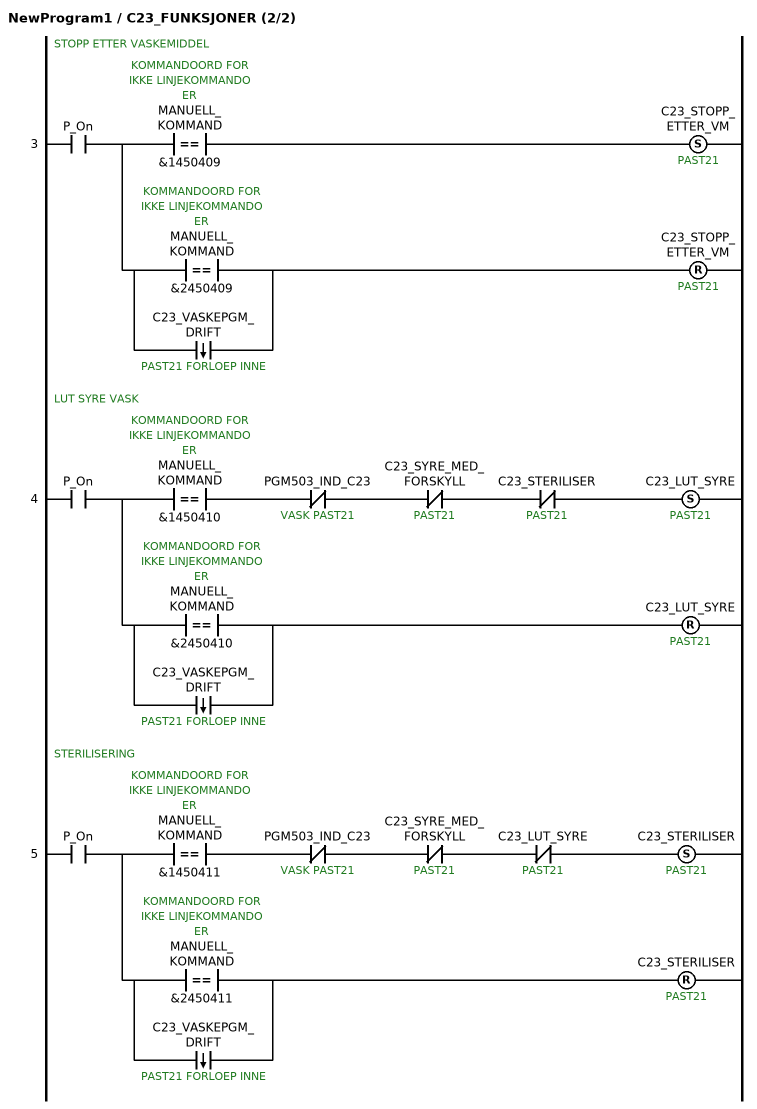
; rung 3: STOPP ETTER VASKEMIDDEL
LD P_On
OUT TR0
AND=L(301) MANUELL_KOMMAND &1450409  ; KOMMANDOORD FOR IKKE LINJEKOMMANDOER
SET C23_STOPP_ETTER_VM  ; PAST21
LD TR0
LD=L(301) MANUELL_KOMMAND &2450409  ; KOMMANDOORD FOR IKKE LINJEKOMMANDOER
%OR C23_VASKEPGM_DRIFT  ; PAST21 FORLOEP INNE
ANDLD
RSET C23_STOPP_ETTER_VM  ; PAST21
; rung 4: LUT SYRE VASK
LD P_On
OUT TR0
AND=L(301) MANUELL_KOMMAND &1450410  ; KOMMANDOORD FOR IKKE LINJEKOMMANDOER
ANDNOT PGM503_IND_C23  ; VASK PAST21
ANDNOT C23_SYRE_MED_FORSKYLL  ; PAST21
ANDNOT C23_STERILISER  ; PAST21
SET C23_LUT_SYRE  ; PAST21
LD TR0
LD=L(301) MANUELL_KOMMAND &2450410  ; KOMMANDOORD FOR IKKE LINJEKOMMANDOER
%OR C23_VASKEPGM_DRIFT  ; PAST21 FORLOEP INNE
ANDLD
RSET C23_LUT_SYRE  ; PAST21
; rung 5: STERILISERING
LD P_On
OUT TR0
AND=L(301) MANUELL_KOMMAND &1450411  ; KOMMANDOORD FOR IKKE LINJEKOMMANDOER
ANDNOT PGM503_IND_C23  ; VASK PAST21
ANDNOT C23_SYRE_MED_FORSKYLL  ; PAST21
ANDNOT C23_LUT_SYRE  ; PAST21
SET C23_STERILISER  ; PAST21
LD TR0
LD=L(301) MANUELL_KOMMAND &2450411  ; KOMMANDOORD FOR IKKE LINJEKOMMANDOER
%OR C23_VASKEPGM_DRIFT  ; PAST21 FORLOEP INNE
ANDLD
RSET C23_STERILISER  ; PAST21
; rung 6: Ingen_kommentar_funnet

### Section C23_TEMP_OVERVÅKING

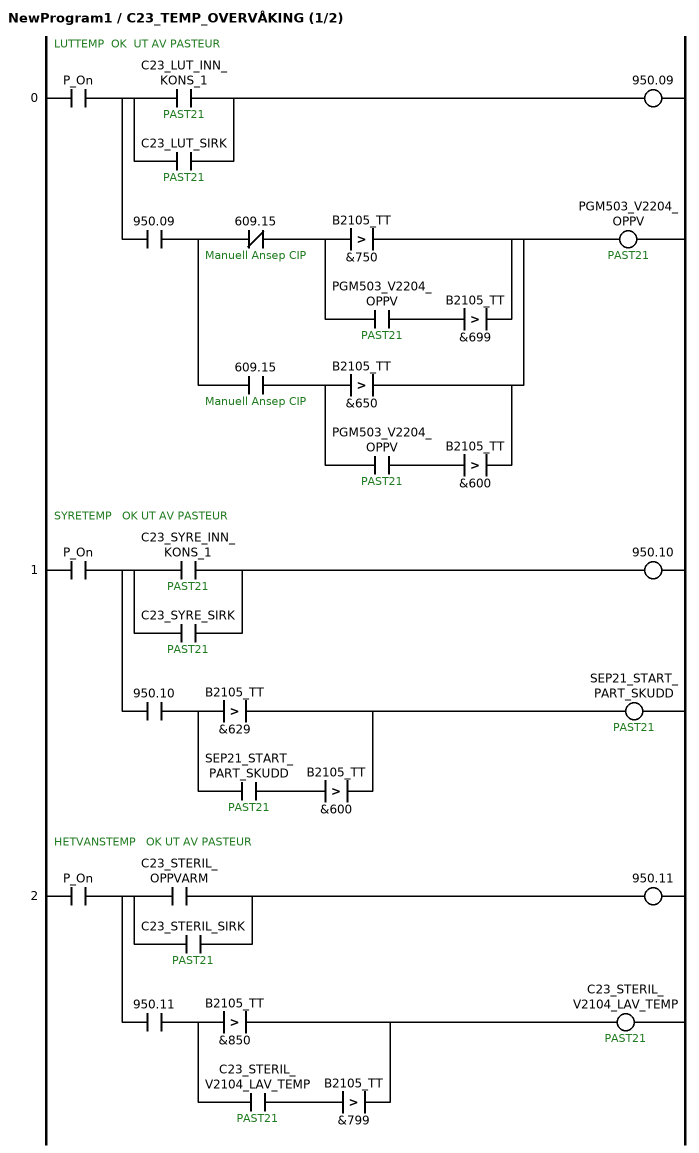
; rung 0: LUTTEMP  OK  UT AV PASTEUR
LD P_On
OUT TR0
LD C23_LUT_INN_KONS_1  ; PAST21
OR C23_LUT_SIRK  ; PAST21
ANDLD
OUT 950.09
LD TR0
AND 950.09
LDNOT 609.15  ; Manuell Ansep CIP
LD>(320) B2105_TT &750
LD PGM503_V2204_OPPV  ; PAST21
AND>(320) B2105_TT &699
ORLD
ANDLD
LD 609.15  ; Manuell Ansep CIP
LD>(320) B2105_TT &650
LD PGM503_V2204_OPPV  ; PAST21
AND>(320) B2105_TT &600
ORLD
ANDLD
ORLD
ANDLD
OUT PGM503_V2204_OPPV  ; PAST21
; rung 1: SYRETEMP   OK UT AV PASTEUR
LD P_On
OUT TR0
LD C23_SYRE_INN_KONS_1  ; PAST21
OR C23_SYRE_SIRK  ; PAST21
ANDLD
OUT 950.10
LD TR0
AND 950.10
LD>(320) B2105_TT &629
LD SEP21_START_PART_SKUDD  ; PAST21
AND>(320) B2105_TT &600
ORLD
ANDLD
OUT SEP21_START_PART_SKUDD  ; PAST21
; rung 2: HETVANSTEMP   OK UT AV PASTEUR
LD P_On
OUT TR0
LD C23_STERIL_OPPVARM
OR C23_STERIL_SIRK  ; PAST21
ANDLD
OUT 950.11
LD TR0
AND 950.11
LD>(320) B2105_TT &850
LD C23_STERIL_V2104_LAV_TEMP  ; PAST21
AND>(320) B2105_TT &799
ORLD
ANDLD
OUT C23_STERIL_V2104_LAV_TEMP  ; PAST21

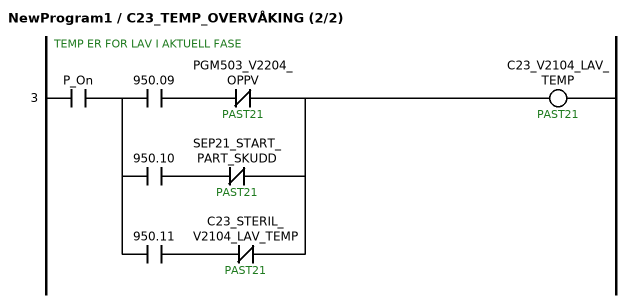
; rung 3: TEMP ER FOR LAV I AKTUELL FASE
LD P_On
LD 950.09
ANDNOT PGM503_V2204_OPPV  ; PAST21
LD 950.10
ANDNOT SEP21_START_PART_SKUDD  ; PAST21
ORLD
LD 950.11
ANDNOT C23_STERIL_V2104_LAV_TEMP  ; PAST21
ORLD
ANDLD
OUT C23_V2104_LAV_TEMP  ; PAST21
; rung 4: Ingen_kommentar_funnet

### Section VST80_C23_TRINN

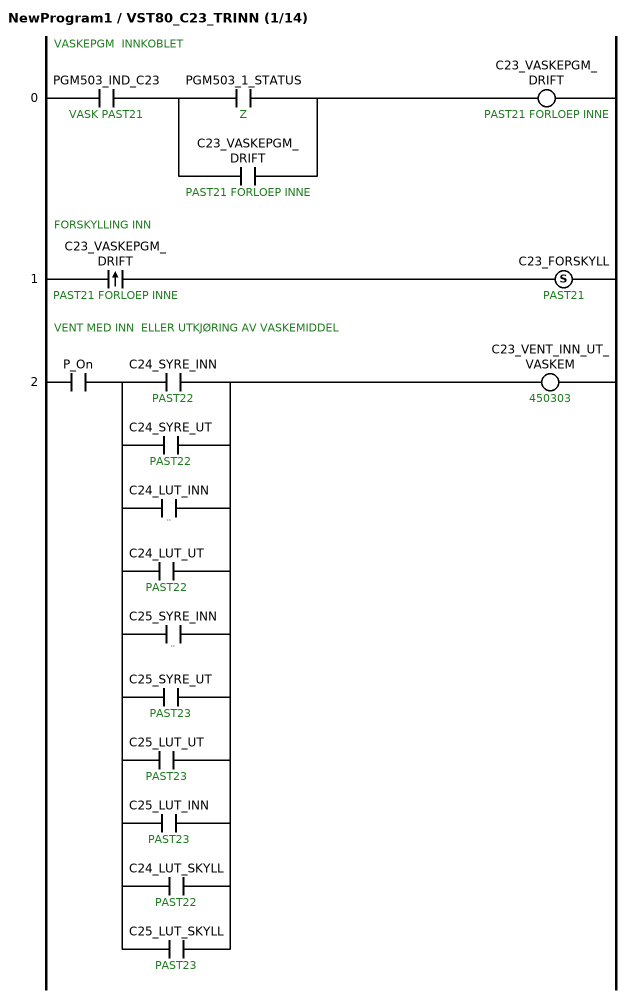
; rung 0: VASKEPGM  INNKOBLET
LD PGM503_IND_C23  ; VASK PAST21
LD PGM503_1_STATUS  ; Z
OR C23_VASKEPGM_DRIFT  ; PAST21 FORLOEP INNE
ANDLD
OUT C23_VASKEPGM_DRIFT  ; PAST21 FORLOEP INNE
; rung 1: FORSKYLLING INN
@LD C23_VASKEPGM_DRIFT  ; PAST21 FORLOEP INNE
SET C23_FORSKYLL  ; PAST21
; rung 2: VENT MED INN  ELLER UTKJØRING AV VASKEMIDDEL
LD P_On
LD C24_SYRE_INN  ; PAST22
OR C24_SYRE_UT  ; PAST22
OR C24_LUT_INN  ; ¨
OR C24_LUT_UT  ; PAST22
OR C25_SYRE_INN  ; ¨
OR C25_SYRE_UT  ; PAST23
OR C25_LUT_UT  ; PAST23
OR C25_LUT_INN  ; PAST23
OR C24_LUT_SKYLL  ; PAST22
OR C25_LUT_SKYLL  ; PAST23
ANDLD
OUT C23_VENT_INN_UT_VASKEM  ; 450303

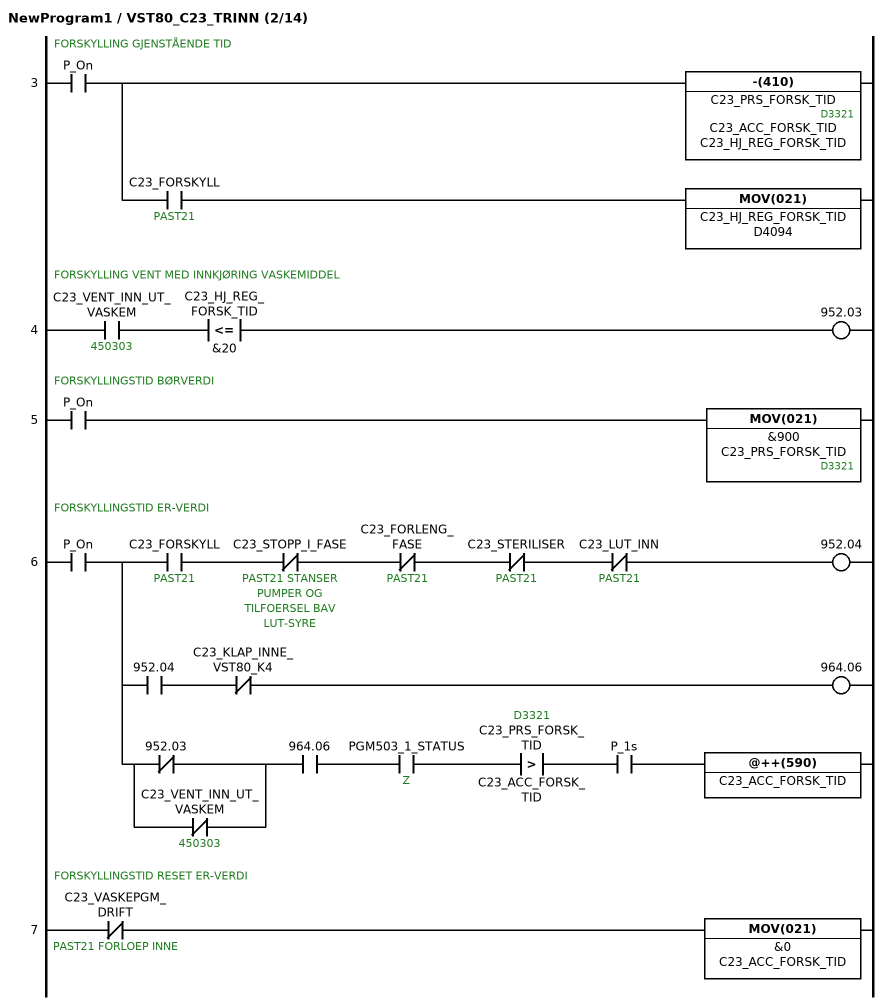
; rung 3: FORSKYLLING GJENSTÅENDE TID
LD P_On
-(410) C23_PRS_FORSK_TID C23_ACC_FORSK_TID C23_HJ_REG_FORSK_TID  ; D3321
AND C23_FORSKYLL  ; PAST21
MOV(021) C23_HJ_REG_FORSK_TID D4094
; rung 4: FORSKYLLING VENT MED INNKJØRING VASKEMIDDEL
LD C23_VENT_INN_UT_VASKEM  ; 450303
AND<=(315) C23_HJ_REG_FORSK_TID &20
OUT 952.03
; rung 5: FORSKYLLINGSTID BØRVERDI
LD P_On
MOV(021) &900 C23_PRS_FORSK_TID  ; D3321
; rung 6: FORSKYLLINGSTID ER-VERDI
LD P_On
OUT TR0
AND C23_FORSKYLL  ; PAST21
ANDNOT C23_STOPP_I_FASE  ; PAST21 STANSER PUMPER OG TILFOERSEL BAV LUT-SYRE
ANDNOT C23_FORLENG_FASE  ; PAST21
ANDNOT C23_STERILISER  ; PAST21
ANDNOT C23_LUT_INN  ; PAST21
OUT 952.04
LD TR0
AND 952.04
ANDNOT C23_KLAP_INNE_VST80_K4
OUT 964.06
LD TR0
LDNOT 952.03
ORNOT C23_VENT_INN_UT_VASKEM  ; 450303
ANDLD
AND 964.06
AND PGM503_1_STATUS  ; Z
AND>(320) C23_PRS_FORSK_TID C23_ACC_FORSK_TID  ; D3321
AND P_1s
@++(590) C23_ACC_FORSK_TID
; rung 7: FORSKYLLINGSTID RESET ER-VERDI
LDNOT C23_VASKEPGM_DRIFT  ; PAST21 FORLOEP INNE
MOV(021) &0 C23_ACC_FORSK_TID

